FUNCTION_BLOCK Detect_Stiction (* Basic FB with empty ECC *)
  (* Standard: 61499-2 *)
  (* Version 1.0, 2020-08-21, Candra Wardaya, UGM *)
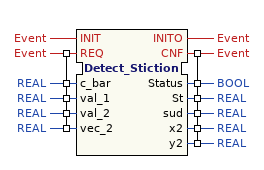
  EVENT_INPUT
    INIT;
    REQ WITH c_bar, val_1, val_2, vec_2;
  END_EVENT
  EVENT_OUTPUT
    INITO;
    CNF WITH Status, St, sud, y2, x2;
  END_EVENT
  VAR_INPUT
    c_bar : REAL;
    val_1 : REAL;
    val_2 : REAL;
    vec_2 : REAL;
  END_VAR
  VAR_OUTPUT
    Status : BOOL;
    St : REAL;
    sud : REAL;
    x2 : REAL;
    y2 : REAL;
  END_VAR
  VAR
    x : REAL; (* Internal Variable *)
    y : REAL; (* Internal Variable *)
    pangkat_x : REAL; (* Internal Variable *)
    pangkat_y : REAL; (* Internal Variable *)
    x1 : REAL; (* Internal Variable *)
    y1 : REAL; (* Internal Variable *)
    x2_y2 : REAL; (* Internal Variable *)
  END_VAR
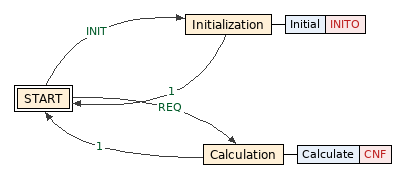
  EC_STATES
    START; (* Initial State *)
    Initialization : Initial -> INITO;
    Calculation : Calculate -> CNF;
  END_STATES
  EC_TRANSITIONS
    START TO Initialization := INIT;
    Initialization TO START := 1;
    START TO Calculation := REQ;
    Calculation TO START := 1;
  END_TRANSITIONS
  ALGORITHM Initial IN ST: (* New Algorithm *)

  END_ALGORITHM
  ALGORITHM Calculate IN ST: (* New Algorithm *)
// m & n // x & y

x1 :=(-c_bar)/val_1;
y1 := (-c_bar)/val_2;

x := SQRT(x1);
y := SQRT(y1);

sud := acos(vec_2);

pangkat_x := (sin(sud))*(sin(sud));
pangkat_y := (cos(sud))*(cos(sud));

x2 := (EXPT(y, 2))*pangkat_x;
y2 := (EXPT(x, 2))*pangkat_y;

IF val_1>0 AND val_2>0 AND c_bar<0 AND x<>y THEN
	Status := TRUE;
	x2_y2 := x2 + y2;
	St := 2*x*y/SQRT(x2_y2);
ELSE
	Status := FALSE;
	St := 0;
END_IF;
  END_ALGORITHM
END_FUNCTION_BLOCK
